// TIA Portal V20 export
TYPE "typeSafetyDoorBox"
// stored: Access Published, IsFailsafeCompliant true, Namespace Safety
   STRUCT
      SI1_Lock_PB : Bool;   // Door Box Lock PB
      SI2_Unlock_PB : Bool;   // Door Box UnLock PB
      SI3_Reset_PB : Bool;   // Door Box Reset PB
   END_STRUCT;
END_TYPE
